Staubli VAL3: onSave.pgx

public program onSave(string& x_sItem[])
  local num i
  local num l_nSize
begin
  //if bToSave
  // update
  if isDefined(pt:tTraj[jEditPoint.sID])
    pt:tTraj[jEditPoint.sID]=jEditPoint
  endIf
  // saveIt
  pt:libSave()
  bToSave=false
  //endIf
end
